Staubli VAL3: Body.dtx

mdesc mNomSpeed
public num nData
